Universal Robots PolyScope program: serve_drink.urp

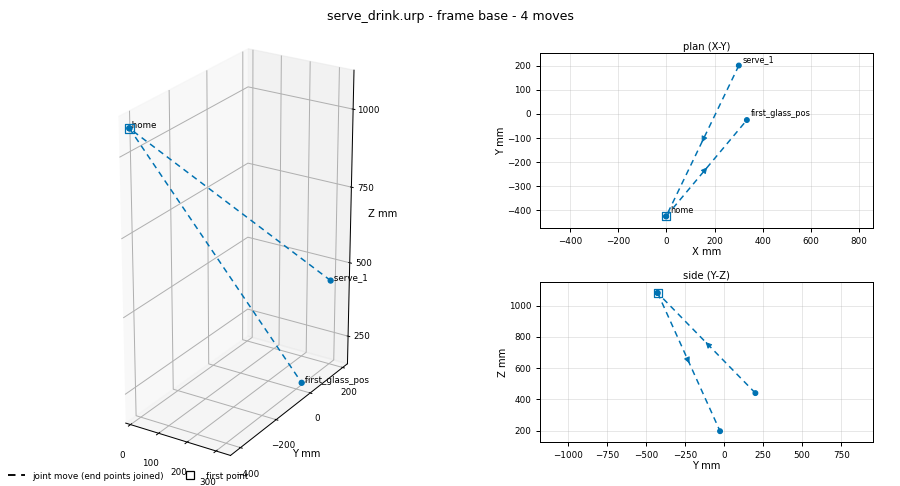
[picture p0: tool path of serve_drink.urp in frame base, 4 of 5 moves have a stored position in this frame; points joined in program order, loops and branches not executed]
Program serve_drink (installation=default directory=/programs/ordering_rfid createdIn=5.9.5.1031259 lastSavedIn=5.12.6.1102099 robotSerialNumber=20215500597)
Calibrated DH parameters: a=[0.000193, -0.066673, -0.391568, -0.000012, 0.00005, 0]; d=[0.162643, -472.05677, 465.132521, 7.058239, 0.099746, 0.099582]; alpha=[1.571116, 0.00089, 0.003862, 1.569269, -1.569248, 0]; deltaTheta=[0, -1.413394, 7.628392, 0.068187, 0, -0.000001]
Robot Program (runOnlyOnce=true)
  MoveJ speed 60 deg/s, acceleration 80 deg/s^2 (useActiveTCP=true) feature=Base
    Waypoint home: TCP in base x=-1.497 y=-424.817 z=1080.554 mm, rx=-0.0043 ry=-2.2185 rz=2.2204 rad; joints [0.002, -90.001, -0.002, -90, -0.001, 0] deg; TCP offset x=0 y=0 z=191.5 mm, rx=0 ry=0 rz=0 rad
  URCap Gripper Activate (Robotiq_Grippers, Robotiq Inc.) dataModel(ResetAndActivateKey=false)
  URCap Gripper (Robotiq_Grippers, Robotiq Inc.) dataModel(position=0.0, force=100.0, speed=100.0, positionInDouble=0.0, forceInDouble=100.0, speedInDouble=100.0, slaveIds=[9], blocking=true)
  glass_pos := [GP_int_in[0],GP_int_in[1]]
  serve_index := GP_int_in[2]
  SuppressedNode
    glass_pos := [1,0]
  SuppressedNode
    serve_index := 3
  MoveJ speed 60 deg/s, acceleration 80 deg/s^2 (useActiveTCP=true) feature=Base
    Waypoint first_glass_pos: TCP in base x=333.528 y=-25.119 z=195.672 mm, rx=1.2266 ry=-2.8464 rz=0.0408 rad; joints [20.899, -65.981, -122.973, -83.466, 88.633, 64.232] deg
  MoveJ speed 60 deg/s, acceleration 80 deg/s^2 (useActiveTCP=true) feature=Base
    offset_pos := p[-0.085*glass_pos[0], -0.075*glass_pos[1],0,0,0,0]
    glass_selected := pose_add(first_glass_pos,offset_pos)
    Waypoint Waypoint (Variable): variable=glass_selected
  MoveL speed 250 mm/s, acceleration 1200 mm/s^2 (useActiveTCP=true) feature=Base
    MoveDirectionNode (selectedDirection=ZMinus)
      Until DISTANCE (allowActions=false deceleration=3 distanceNodeType=STOP) Distance=0.05; motionParameters(blendRadius=0)
    URCap Gripper (Robotiq_Grippers, Robotiq Inc.) dataModel(position=100.0, force=60.0, speed=100.0, positionInDouble=100.0, forceInDouble=60.0, speedInDouble=100.0, slaveIds=[9], blocking=true)
    MoveDirectionNode (selectedDirection=ZPlus)
      Until DISTANCE (allowActions=false deceleration=3 distanceNodeType=STOP) Distance=0.175; motionParameters(blendRadius=0)
  MoveJ speed 60 deg/s, acceleration 80 deg/s^2 (useActiveTCP=true) feature=Base
    Waypoint serve_1: TCP in base x=300.135 y=201.043 z=439.51 mm, rx=-3.0992 ry=-0.1071 rz=0.0083 rad; joints [54.206, -72.445, -83.666, -112.335, 91.901, -39.91] deg; TCP offset x=0 y=0 z=191.5 mm, rx=0 ry=0 rz=0 rad
  move_needed := [5,4,1,0]
  move_times := move_needed[serve_index]
  Loop While (checkContinuously=false) expression=move_times>0
    MoveL speed 250 mm/s, acceleration 1200 mm/s^2 (useActiveTCP=true) feature=Base
      MoveDirectionNode (selectedDirection=XMinus)
        Until DISTANCE (allowActions=false deceleration=3 distanceNodeType=STOP) Distance=0.115; motionParameters(blendRadius=0)
    Script: move_times=move_times-1
  MoveL speed 250 mm/s, acceleration 1200 mm/s^2 (useActiveTCP=true) feature=Base
    MoveDirectionNode (selectedDirection=ZMinus)
      Until DISTANCE (allowActions=false deceleration=3 distanceNodeType=STOP) Distance=0.211; motionParameters(blendRadius=0)
    URCap Gripper (Robotiq_Grippers, Robotiq Inc.) dataModel(position=0.0, force=100.0, speed=50.0, positionInDouble=0.0, forceInDouble=100.0, speedInDouble=50.0, slaveIds=[9], blocking=true)
    MoveDirectionNode (selectedDirection=ZPlus)
      Until DISTANCE (allowActions=false deceleration=3 distanceNodeType=STOP) Distance=0.1; motionParameters(blendRadius=0)
  MoveJ speed 60 deg/s, acceleration 80 deg/s^2 (useActiveTCP=true) feature=Base
    Waypoint home: TCP in base x=-1.497 y=-424.817 z=1080.554 mm, rx=-0.0043 ry=-2.2185 rz=2.2204 rad; joints [0.002, -90.001, -0.002, -90, -0.001, 0] deg; TCP offset x=0 y=0 z=191.5 mm, rx=0 ry=0 rz=0 rad
